// SIMATIC S7-200 project (STEP 7-Micro/WIN), CPU 224 REL 02.01

SYMBOL_TABLE USR1
pre_l            VD46
pre_r            VD42
before           VD16
set4             VD12
set3             VD8
set2             VD4
set1             VD0
retur            Q1.1
ascent           Q1.0
discharge        Q0.7
alarm            Q0.4
l                Q0.2
r                Q0.1
high             Q0.0
len              VD20
re               M0.3
work             M0.2
le               M0.1
find             M0.0
set              I1.5
left             I1.4
b                I1.2
a                I1.1
zero             I1.0
mstart           I0.5
mreturn          I0.4
m                I0.3
stop             I0.2
return           I0.1
start            I0.0
find_r           M0.4
find_l           M0.5
re_r             M0.6
re_l             M0.7
work_r           M1.0
work_l           M1.1
re_high          M1.2
work_high        M1.3
m_r              M1.4
m_l              M1.5
pulse_n1         VD28
pot0             VW36
pulse_n2         VD32
len_loc          VD38
ko_r             M1.6
ko_l             M1.7
overflow_r       M2.0
overflow_l       M2.1
END_SYMBOL_TABLE

ORGANIZATION_BLOCK MAIN:OB1
TITLE=工业流水线中用于物料搬运的水平小车的自动化控制程序。小车通过高速计数器精确记录位置。
// 系统通过模式切换判断当前模式。在手动模式下，只有按下手动启动按钮或手动返回按钮，小车才会向右或向左移动。当按下返回原点按钮时，系统设置返回原点标志，根据高速计数器与零的比较，激活向右返回或向左返回，并在接近原点时通过高速返回提高效率。到达原点后，原点传感器触发。在手动模式下通过设置按钮保存高速计数器的当前值到设定值中。向右移动输出控制小车向右移动。向左移动输出控制小车向左移动。高速移动输出实现小车高低速切换。小车移动时，高速计数器的值超出预设右值或预设左值时，触发溢出标志。在自动模式下，向右移动输出或向左移动输出激活但高速计数器未变化时，触发报警输出。报警通过按下启动按钮复位。
BEGIN
Network 1 // NETWORK TITLE (single line)
//  
// NETWORK COMMENTS
//  
// 
LD     SM0.1
MOVB   16#FC, SMB47
HDEF   1, 10
MOVD   +0, SMD48
HSC    1
Network 2
LD     SM0.0
BTI    SMB28, pot0:VW36
MOVW   pot0:VW36, VW30
MUL    +4, pulse_n1:VD28
MOVD   0, pulse_n2:VD32
-D     pulse_n1:VD28, pulse_n2:VD32
Network 3
LD     start:I0.0
O      find:M0.0
AN     alarm:Q0.4
AN     m:I0.3
AN     re:M0.3
AN     work:M0.2
AN     stop:I0.2
AN     zero:I1.0
LPS
=      find:M0.0
AN     le:M0.1
AN     l:Q0.2
=      find_r:M0.4
LPP
LD     left:I1.4
O      le:M0.1
ALD
=      le:M0.1
TON    T37, +5
A      T37
AN     r:Q0.1
=      find_l:M0.5
Network 4
LDN    a:I1.1
AN     b:I1.2
CALL   SBR_0:SBR0, set1:VD0
A      m:I0.3
A      set:I1.5
MOVD   HC1, set1:VD0
Network 5
LD     a:I1.1
AN     b:I1.2
CALL   SBR_0:SBR0, set2:VD4
A      m:I0.3
A      set:I1.5
MOVD   HC1, set2:VD4
Network 6
LDN    a:I1.1
A      b:I1.2
CALL   SBR_0:SBR0, set3:VD8
A      m:I0.3
A      set:I1.5
MOVD   HC1, set3:VD8
Network 7
LD     a:I1.1
A      b:I1.2
CALL   SBR_0:SBR0, set4:VD12
A      m:I0.3
A      set:I1.5
MOVD   HC1, set4:VD12
Network 8
LD     return:I0.1
O      re:M0.3
AN     stop:I0.2
AN     m:I0.3
AN     alarm:Q0.4
AN     zero:I1.0
AN     find:M0.0
AN     work:M0.2
LPS
=      re:M0.3
LDD>   HC1, +0
O      re_l:M0.7
ALD
AN     re_r:M0.6
=      re_l:M0.7
LRD
LDD<   HC1, +0
O      re_r:M0.6
ALD
AN     re_l:M0.7
=      re_r:M0.6
LPP
LDD>=  HC1, pulse_n1:VD28
OD<=   HC1, pulse_n2:VD32
ALD
=      re_high:M1.2
Network 9
LD     m:I0.3
LPS
AN     l:Q0.2
A      mstart:I0.5
=      m_r:M1.4
LPP
AN     r:Q0.1
A      mreturn:I0.4
=      m_l:M1.5
Network 10
LDN    m:I0.3
LD     r:Q0.1
O      l:Q0.2
ALD
LPS
A      T39
AD=    HC1, before:VD16
S      alarm:Q0.4, 1
LPP
AN     T39
LPS
EU
MOVD   HC1, before:VD16
LPP
TON    T39, +20
Network 11
LD     start:I0.0
AN     m:I0.3
A      alarm:Q0.4
R      alarm:Q0.4, 1
Network 12
LD     find_r:M0.4
O      re_r:M0.6
O      work_r:M1.0
O      m_r:M1.4
AN     stop:I0.2
=      r:Q0.1
=      ascent:Q1.0
Network 13
LD     find_l:M0.5
O      re_l:M0.7
O      work_l:M1.1
O      m_l:M1.5
AN     stop:I0.2
=      l:Q0.2
=      retur:Q1.1
Network 14
LD     work_high:M1.3
O      re_high:M1.2
AN     stop:I0.2
=      high:Q0.0
END_ORGANIZATION_BLOCK

SUBROUTINE_BLOCK SBR_0:SBR0
TITLE= 
// SUBROUTINE COMMENTS
// Press F1 for help and example program
//  
VAR_INPUT
setv:DWORD;	// LD0 
END_VAR
BEGIN
Network 1 // NETWORK TITLE (single line)
//  
// NETWORK COMMENTS
//  
// 
LD     zero:I1.0
A      start:I0.0
O      work:M0.2
LPS
AN     stop:I0.2
AN     alarm:Q0.4
AN     m:I0.3
AN     find:M0.0
AN     re:M0.3
AN     return:I0.1
=      work:M0.2
LRD
MOVD   #setv:LD0, len:VD20
-D     HC1, len:VD20
LRD
AD>=   len:VD20, pre_r:VD42
=      work_r:M1.0
LRD
AD<=   len:VD20, pre_l:VD46
=      work_l:M1.1
LRD
LDD<=  len:VD20, pulse_n2:VD32
OD>=   len:VD20, pulse_n1:VD28
ALD
=      work_high:M1.3
LRD
AD<    len:VD20, +50
AD>    len:VD20, -50
LPS
AN     work_l:M1.1
AN     work_r:M1.0
TON    T38, +5
LPP
AN     zero:I1.0
A      T38
=      discharge:Q0.7
LRD
LD     work_high:M1.3
A      work_r:M1.0
O      ko_r:M1.6
AN     work_l:M1.1
ALD
=      ko_r:M1.6
A      discharge:Q0.7
EU
MOVD   len:VD20, len_loc:VD38
AENO
/D     +2, len_loc:VD38
AENO
-D     len_loc:VD38, pre_r:VD42
LRD
LD     work_high:M1.3
A      work_l:M1.1
O      ko_l:M1.7
AN     work_r:M1.0
ALD
=      ko_l:M1.7
A      discharge:Q0.7
EU
MOVD   len:VD20, len_loc:VD38
AENO
/D     +2, len_loc:VD38
AENO
-D     len_loc:VD38, pre_l:VD46
LRD
LD     work_high:M1.3
A      work_r:M1.0
O      overflow_r:M2.0
AN     discharge:Q0.7
ALD
=      overflow_r:M2.0
A      work_l:M1.1
EU
+D     10, pre_r:VD42
LRD
LD     work_high:M1.3
A      work_l:M1.1
O      overflow_l:M2.1
AN     discharge:Q0.7
ALD
=      overflow_l:M2.1
A      work_r:M1.0
EU
+D     -10, pre_l:VD46
LPP
LPS
AD<    pre_r:VD42, 5
MOVD   5, pre_r:VD42
LRD
AD>    pre_l:VD46, -5
MOVD   -5, pre_l:VD46
LRD
AD>    pre_r:VD42, 70
MOVD   50, pre_r:VD42
LPP
AD<    pre_l:VD46, -70
MOVD   -50, pre_l:VD46
END_SUBROUTINE_BLOCK

DATA_BLOCK_TAB USER1
BEGIN
//DATA BLOCK COMMENTS
         set1, 0
         set2, 0
         set3, 0
         set4, 0
         before, 0
         len, 0
         pulse_n1
         pulse_n2, 0
         pot0, 0
         len_loc, 0
         pre_r, 30
         pre_l, -30
//Press F1 for help and example data block
END_DATA_BLOCK_TAB
